RoboDK station: Coursework2_robot_manipulator.rdk

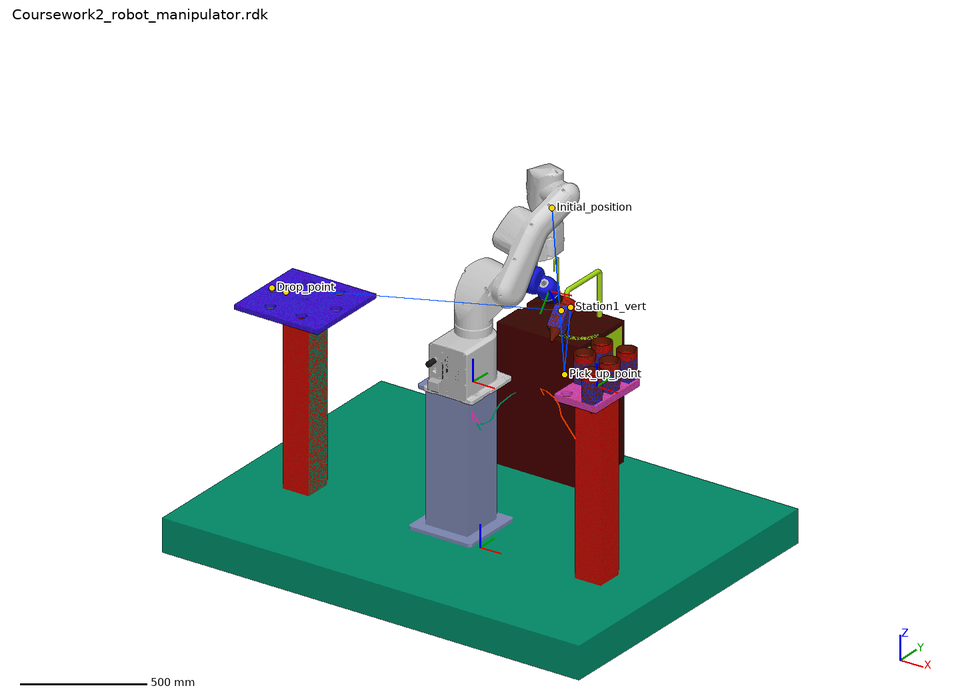
[picture v0: the station drawn from its stored meshes, robots at their saved joint values, targets as dots, program paths as lines]
Station Coursework2_robot_manipulator (saved by RoboDK 5.8.0). Poses are relative to the parent item; angles as X-Y-Z fixed-axis rotations.
  - frame baseframe at (0, 0, 0) mm
    - object PDE4431_CW2_2024 at (0, 0, 0) mm, rotated rx 90 ry 0 rz 0 deg, size 2000 x 980 x 1500 mm, geometry from PDE4431_CW2_2024.STEP
    - frame Epson VT6 Base at (45, -110, 780) mm
      - robot Epson VT6: 6 axes, payload 6 kg, reach 920 mm, repeatability 0.1 mm, weight 40 kg
          modified DH rows (alpha deg, a mm, theta deg, d mm): 0, 0, 0, 412; -90, 100, -90, 0; 0, 420, 0, 0; -90, 0, 0, 400; 90, 0, 0, 0; -90, 0, 0, 80
          base shift (0, 0, 0) mm, rotated rx 0 ry 0 rz 90 deg
          joint limits [-170, -160, -51, -200, -125, -360] to [170, 65, 190, 200, 125, 360]; home [0, 0, 0, 0, 0, 0]; saved at [-14.215, -42.735, -50.612, -158.07, -43.09, 91.944]
        - tool Tool 1, TCP at (0, 0, 180) mm, rotated rx -90 ry 0 rz 0 deg
          - object Cone-Part at (0, -10, 30) mm, rotated rx -90 ry 0 rz 180 deg, size 84.9 x 182 x 85 mm, geometry from Cone-Part.STEP
        - frame RobotiQ 2F-140 Gripper (Mechanism) Base at (0, 0, 0) mm
          - robot RobotiQ 2F-140 Gripper (Mechanism) (model RobotiQ 2F140): 1 axes, payload 5 kg
              joint limits [0] to [140]; home [140]; saved at [90]
    - frame input_area_reference_frame at (700, -200, 980) mm
      - object Cone-Part at (60, 120, 50) mm, rotated rx 90 ry 0 rz 90 deg, size 84.9 x 182 x 85 mm, geometry from Cone-Part.STEP
      - object Cone-Part at (-60, 120, 50) mm, rotated rx 90 ry 0 rz 90 deg, size 84.9 x 182 x 85 mm, geometry from Cone-Part.STEP
      - object Cone-Part at (60, 0, 50) mm, rotated rx 90 ry 0 rz 90 deg, size 84.9 x 182 x 85 mm, geometry from Cone-Part.STEP
      - object Cone-Part at (60, -120, 50) mm, rotated rx 90 ry 0 rz 90 deg, size 84.9 x 182 x 85 mm, geometry from Cone-Part.STEP
      - object Cone-Part at (-60, 0, 50) mm, rotated rx 90 ry 0 rz 90 deg, size 84.9 x 182 x 85 mm, geometry from Cone-Part.STEP
    - target Initial_position (Cartesian target) at (0, 493.22, 1288.03) mm, rotated rx 138 ry 0 rz 0 deg; joints [0, 0, 0, 0, -42, -90] of Epson VT6
    - target Gripper_open (Cartesian target) at (0.67, 380.04, 1461.97) mm, rotated rx -90 ry 0 rz 0 deg; joints [90, -0.57, 0.57, -89.99, -12.6, 0] of RobotiQ 2F-140 Gripper (Mechanism)
    - target Gripper_closed (Cartesian target) at (0.67, 380.04, 1461.97) mm, rotated rx -90 ry 0 rz 0 deg; joints [60, -0.57, 0.57, -89.99, -12.6, 0] of RobotiQ 2F-140 Gripper (Mechanism)
    - target Pick_up_point (Cartesian target) at (630, -320, 1060) mm, rotated rx 180 ry 0 rz -90 deg; joints [-107.969, 3.021, -41.964, -152.706, -42.282, 69.105] of Epson VT6
    - target Station1_vert (joint target) at (117.17, 455.58, 902) mm, rotated rx -180 ry 0 rz 9.17 deg; joints [-20.193, -81.214, -36.487, -147.565, -113.899, 104.438] of Epson VT6
    - target station1_return (joint target) at (107.17, 405.58, 902) mm, rotated rx 130 ry 0 rz 9.17 deg; joints [-14.215, -42.735, -50.612, -158.07, -43.09, 91.944] of Epson VT6
    - target Drop_point (joint target) at (-765.8, -330, 1052.5) mm, rotated rx -180 ry 0 rz 90 deg; joints [111.773, -56.2, -12.685, -23.179, 70.455, -81.848] of Epson VT6
    - object Pedestal_4 at (0, -130, 150) mm, rotated rx 90 ry 0 rz 0 deg, size 300 x 630 x 300 mm, geometry from Pedestal_4.STEP
    - target Target 8 (Cartesian target) at (-700.8, -330, 1052.5) mm, rotated rx -180 ry 0 rz 90 deg; joints [114.364, -53.634, -22.613, -24.996, 77.493, -84.235] of Epson VT6
    - target Target 9 (Cartesian target) at (-700.8, -330, 1052.5) mm, rotated rx -180 ry 0 rz 90 deg; joints [114.364, -53.634, -22.613, -24.996, 77.493, -84.235] of Epson VT6
  - program Gripper_open (1 instructions, listed below)
  - program Gripper_close (1 instructions, listed below)
  - program Test1 (13 instructions, listed below)
  - program Prog4 (1 instructions, listed below)
  - object Curve1 at (0, 0, 832) mm, geometry from Imported curve
  - machining project Cone_curve_Station_1: rotz(0) | rotx(0)*rotY(0) | onStart | onPathStart | onApproach | onPoint | onRetract | onFinish | SetRPM(%1) | SetTool(%1) | Extruder(%1) | default | default | OutOnMov(%1) | OutOffMov(%1) | onPathFinish | M_RunCode(%1)
  - object Curve2 at (0, 0, 832) mm, geometry from 000000
  - machining project Path2 settings: rotZ(0) | rotX(0)*rotY(0) | onStart | onPathStart | onApproach | onPoint | onRetract | onFinish | SetRPM(%1) | SetTool(%1) | Extruder(%1) | default | default | OutOnMov(%1) | OutOffMov(%1) | onPathFinish | M_RunCode(%1)
  - object Curve3 at (0, 0, 832) mm
  - machining project Path3 settings: rotZ(0) | rotX(0)*rotY(0) | onStart | onPathStart | onApproach | onPoint | onRetract | onFinish | SetRPM(%1) | SetTool(%1) | Extruder(%1) | default | default | OutOnMov(%1) | OutOffMov(%1) | onPathFinish | M_RunCode(%1)
  - Python program Prog8 (listed below)
  - program Cone_curve_Station_1 (17 instructions, listed below)
  - program Path2 (23 instructions, listed below)
  - program Path3 (16 instructions, listed below)
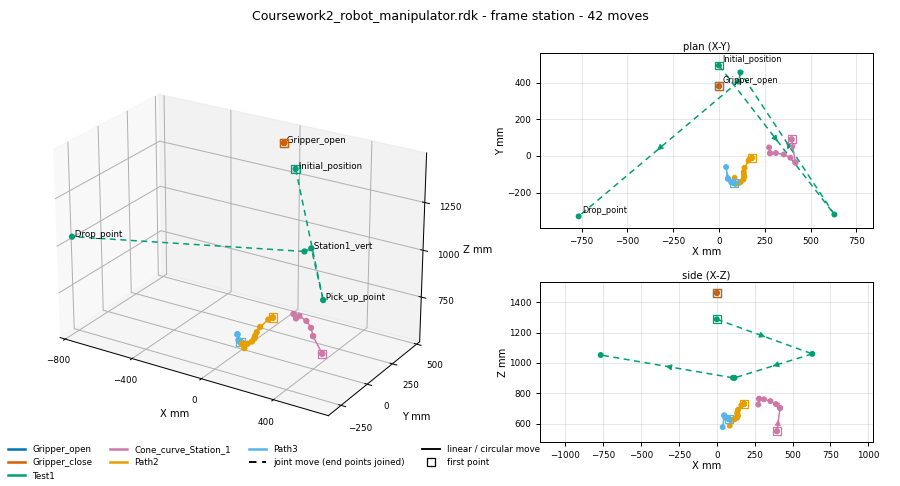
[picture p0: tool path of Coursework2_robot_manipulator.rdk in frame station, 42 of 42 moves have a stored position in this frame; points joined in program order, loops and branches not executed]

--- program Gripper_open (robot RobotiQ 2F-140 Gripper (Mechanism)) ---
  MoveJ (Gripper_open)

--- program Gripper_close (robot RobotiQ 2F-140 Gripper (Mechanism)) ---
  MoveJ (Gripper_closed)

--- program Test1 (robot Epson VT6) ---
  Set Ref.: baseframe
  MoveJ (Initial_position)
  Call Gripper_open
  MoveJ (Target 4) -> target Pick_up_point
  Call Gripper_close
  Attach to Tool 1
  Call Cone_curve_Station_1
  MoveJ (Station1_vert)
  MoveJ (station1_return)
  Call Path2
  Call Path3
  MoveJ (Drop_point)
  Call Gripper_open

--- program Prog4 (robot Epson VT6) ---
  Replace objects

--- Python program Prog8 ---
from robodk.robolink import *
from robodk.robomath import *
import time

#Connection b/w roboDK
RDK=Robolink()

#conf. robot
robot=RDK.Item('Epson VT6')

robot.setSpeed(200)

#setting Target
home = RDK.Item('Initial_position')

#Pick_up_points with one point reference
pickup1=RDK.Item('Pick_up_point')
pickup2=pickup1.Pose()*transl(-120,0,0)
pickup3=pickup1.Pose()*transl(-240,0,0)
pickup4=pickup1.Pose()*transl(0,-120,0)
pickup5=pickup1.Pose()*transl(-120,-120,0)
pickup6=pickup1.Pose()*transl(-240,-120,0)

#Drop_points with one point reference
drop1=RDK.Item('Drop_point')
drop2=drop1.Pose()*transl(129.9,-75,0)
drop3=drop1.Pose()*transl(259.8,0,0)
drop4=drop1.Pose()*transl(0,150,0)
drop5=drop1.Pose()*transl(129.9,225,0)
drop6=drop1.Pose()*transl(259.8,150,0)


robot.MoveJ(home)
robot.MoveJ(drop6)

--- program Cone_curve_Station_1 (robot Epson VT6) ---
  Smooth(1)
  Set speed (1000.0 mm/s)
  Set Ref.: RobotiQ 2F-140 Gripper (Mechanism) Base
  Set Tool: Tool 1
  Show Tool 1
  MoveJ 1 to (235.67, 499.97, 220) mm, rotated rx 130 ry 0 rz 60.63 deg; joints [-32.495, -35.422, -9.628, -48.591, -58.845, 34.479]
  MoveL 2 to (235.67, 499.97, 220) mm, rotated rx 130 ry 0 rz 60.63 deg; joints [-32.495, -35.422, -9.628, -48.591, -58.845, 34.479]
  MoveL 3 to (235.67, 499.97, 20) mm, rotated rx 130 ry 0 rz 60.63 deg; joints [-32.495, -58.155, -6.814, -60.99, -47.215, 54.854]
  MoveL 4 to (235.67, 499.97, 20) mm, rotated rx 130 ry 0 rz 60.63 deg; joints [-32.495, -58.155, -6.814, -60.99, -47.215, 54.854]
  Set speed (50.0 mm/s)
  MoveL 5 to (213.11, 459.87, 20) mm, rotated rx 130 ry 0 rz 42.48 deg; joints [-32.175, -53.633, -23.445, -89.489, -38.309, 69.642]
  MoveL 6 to (179.87, 429.44, 20) mm, rotated rx 130 ry 0 rz 24.5 deg; joints [-27.795, -51.909, -37.041, -126.693, -39.365, 88.69]
  MoveL 7 to (138.68, 410.66, 20) mm, rotated rx 130 ry 0 rz 9.17 deg; joints [-18.69, -52.635, -45.751, -155.976, -47.548, 95.3]
  MoveL 8 to (107.17, 405.58, 20) mm, rotated rx 130 ry 0 rz 9.17 deg; joints [-14.215, -53.09, -47.595, -160.533, -49.956, 95.516]
  Set speed (1000.0 mm/s)
  MoveL 9 to (107.17, 405.58, 20) mm, rotated rx 130 ry 0 rz 9.17 deg; joints [-14.215, -53.09, -47.595, -160.533, -49.956, 95.516]
  MoveL 10 to (107.17, 405.58, 70) mm, rotated rx 130 ry 0 rz 9.17 deg; joints [-14.215, -42.735, -50.612, -158.07, -43.09, 91.944]

--- program Path2 (robot Epson VT6) ---
  Smooth(1)
  Set speed (1000.0 mm/s)
  Set Ref.: RobotiQ 2F-140 Gripper (Mechanism) Base
  Set Tool: Tool 1
  Show Tool 1
  MoveJ 1 to (4.44, 434.85, 40) mm, rotated rx 130 ry 0 rz -37.79 deg; joints [19.104, -48.457, -38.321, 119.728, -38.319, -265.644]
  MoveL 2 to (4.44, 434.85, 40) mm, rotated rx 130 ry 0 rz -37.79 deg; joints [19.104, -48.457, -38.321, 119.728, -38.319, -265.644]
  MoveL 3 to (4.44, 434.85, 40) mm, rotated rx 130 ry 0 rz -37.79 deg; joints [19.104, -48.457, -38.321, 119.728, -38.319, -265.644]
  MoveL 4 to (4.44, 434.85, 40) mm, rotated rx 130 ry 0 rz -37.79 deg; joints [19.104, -48.457, -38.321, 119.728, -38.319, -265.644]
  Set speed (50.0 mm/s)
  MoveL 5 to (-14.66, 449.66, 40) mm, rotated rx 130 ry 0 rz -58.41 deg; joints [23.166, -50.219, -26.667, 82.641, -39.877, -249.508]
  MoveL 6 to (-42.76, 495.36, 40) mm, rotated rx 130 ry 0 rz -74.77 deg; joints [23.918, -54.966, -9.837, 56.916, -49.321, -236.292]
  MoveL 7 to (-50.7, 524.53, 40) mm, rotated rx 130 ry 0 rz -84.24 deg; joints [22.981, -58.691, 0.728, 47.241, -56.742, -232.705]
  MoveL 8 to (-52.73, 544.68, 40) mm, rotated rx 130 ry 0 rz -90.49 deg; joints [21.982, -61.509, 8.097, 42.25, -62.055, -231.428]
  MoveL 9 to (-52.65, 554.44, 40) mm, rotated rx 130 ry 0 rz -99.88 deg; joints [20.728, -64.435, 15.394, 36.439, -68.656, -232.719]
  MoveL 10 to (-51.8, 559.3, 40) mm, rotated rx 130 ry 0 rz -67.84 deg; joints [22.537, -57.658, -2.086, 58.775, -48.734, -227.908]
  MoveL 11 to (-58.92, 576.77, 40) mm, rotated rx 130 ry 0 rz -39.55 deg; joints [20.657, -53.944, -12.994, 89.358, -33.909, -232.455]
  MoveL 12 to (-76.79, 591.52, 40) mm, rotated rx 130 ry 0 rz -23.9 deg; joints [19.052, -53.111, -15.694, 110.258, -27.833, -238.151]
  MoveL 13 to (-85.16, 595.24, 40) mm, rotated rx 130 ry 0 rz -5.76 deg; joints [15.249, -52.044, -19.375, 144.64, -23.462, -253.329]
  MoveL 14 to (-105.32, 597.27, 40) mm, rotated rx 130 ry 0 rz -5.76 deg; joints [17.163, -52.4, -18.113, 140.4, -23.123, -250.682]
  Set speed (1000.0 mm/s)
  MoveL 15 to (-105.32, 597.27, 40) mm, rotated rx 130 ry 0 rz -5.76 deg; joints [17.163, -52.4, -18.113, 140.4, -23.123, -250.682]
  MoveL 16 to (-105.32, 597.27, 90) mm, rotated rx 130 ry 0 rz -5.76 deg; joints [17.163, -45.707, -19.841, 131.55, -19.541, -241.189]

--- program Path3 (robot Epson VT6) ---
  Smooth(1)
  Set speed (1000.0 mm/s)
  Set Ref.: RobotiQ 2F-140 Gripper (Mechanism) Base
  Set Tool: Tool 1
  Show Tool 1
  MoveJ 1 to (-115.1, 588.73, 40) mm, rotated rx 130 ry 0 rz 14.39 deg; joints [12.455, -51.647, -20.832, -176.753, -22.495, 88.48]
  MoveL 2 to (-115.1, 588.73, 40) mm, rotated rx 130 ry 0 rz 14.39 deg; joints [12.455, -51.647, -20.832, -176.753, -22.495, 88.48]
  MoveL 3 to (-115.1, 588.73, 40) mm, rotated rx 130 ry 0 rz 14.39 deg; joints [12.455, -51.647, -20.832, -176.753, -22.495, 88.48]
  MoveL 4 to (-115.1, 588.73, 40) mm, rotated rx 130 ry 0 rz 14.39 deg; joints [12.455, -51.647, -20.832, -176.753, -22.495, 88.48]
  Set speed (50.0 mm/s)
  MoveL 5 to (-116.49, 588.38, 40) mm, rotated rx 130 ry 0 rz 31.56 deg; joints [7.582, -52.149, -19, -139.719, -23.834, 71.035]
  MoveL 6 to (-127.34, 581.71, 40) mm, rotated rx 130 ry 0 rz 63.07 deg; joints [2.169, -55.1, -9.431, -85.194, -34.309, 48.192]
  MoveL 7 to (-141.71, 553.41, 40) mm, rotated rx 130 ry 0 rz 63.07 deg; joints [3.671, -53.55, -14.255, -91.403, -33.605, 54.019]
  Set speed (1000.0 mm/s)
  MoveL 8 to (-141.71, 553.41, 40) mm, rotated rx 130 ry 0 rz 63.07 deg; joints [3.671, -53.55, -14.255, -91.403, -33.605, 54.019]
  MoveL 9 to (-141.71, 553.41, 140) mm, rotated rx 130 ry 0 rz 63.07 deg; joints [3.671, -40.938, -16.763, -76.505, -34.681, 36.065]
